PROGRAM PRG_SystemControlMachineWork
VAR
	bFirstCycle		: BOOL;
END_VAR

IF (GVL_SystemVariable.bDefaultInitDone AND
	GVL_SystemVariable.bMachineInitDone) THEN
	;
	(*	Wywołanie obsługi Logera	*)
	GVL_SystemVariable.fbLogger ();
	(*	Wywołanie pracy maszyny		*)
	GVL_SystemVariable.fbMachineControl ();
END_IF

END_PROGRAM

(* stored: Version 1.1.0.1
   POU PRG_SystemControlMachineWork: Id {7cf4e122-3b89-4f4f-9f5d-2b648ff60401}, SpecialFunc None *)
